TYPE ST_ReadAllOffsetDateStatus EXTENDS ST_StatusBasic :
STRUCT
END_STRUCT
END_TYPE

(* stored: Version 1.1.0.1, ProductVersion 3.1.4024.13
   DUT ST_ReadAllOffsetDateStatus: Id {f2d05a01-5133-475f-9765-9321402fa928} *)
